(* Logix 5000 project; controller inz_PD_LK vendor 1 type 14 code 285 rev 34.11; software revision 34.01 *)

TASK MainTask (continuous, watchdog 500 ms) : Paleczka_silnik, Dzwonki_silnik, Paleczka_note_move, Dzwonki_belt_move, buttons, status, TIMER, Lights

MODULES
   Local : vendor 1 type 14 code 285 (5069 0, rev 34.11)
      serwowzmacniacz : vendor 1 type 45 code 1 (Ethernet 192.168.1.26, rev 5.2, AMotionDiagnostics RPI 1 ms)
      serwowzmacniacz2 : vendor 1 type 45 code 1 (Ethernet 192.168.1.27, rev 5.2, AMotionDiagnostics RPI 1 ms)
      Input : 5069-IB16 (5069 1, rev 2.1, StandardDataDriven RPI 5 ms)
      Output : 5069-OB16 (5069 2, rev 3.1, StandardDataDriven RPI 5 ms)
END_MODULES

VAR_GLOBAL   (* controller tags *)
   all_rise : BOOL;
   auto_mode : ALIAS FOR Local:1:I.Pt11.Data;
   belt_button : ALIAS FOR Local:1:I.Pt02.Data;
   belt_degree : DINT := 28;
   D_JOG_Axis_OFF : BOOL := 1;
   D_JOG_Axis_ON : BOOL;
   D_motor_start : BOOL;
   D_motor_stop : BOOL := 1;
   degree : DINT := -20;
   Dzwonki : AXIS_CIP_DRIVE;
   Estop_button : ALIAS FOR Local:1:I.Pt00.Data;
   forced_OFF : BOOL;
   forced_ON : BOOL := 1;
   green_lamp : ALIAS FOR Local:2:O.Pt13.Data;
   L_R_switch : ALIAS FOR Local:1:I.Pt10.Data;
   Motion : MOTION_GROUP;
   MotionControlMAFR_D : MOTION_INSTRUCTION := (FLAGS := 570425344, DN := 1, STATE := 1);
   MotionControlMAFR_P : MOTION_INSTRUCTION := (FLAGS := 570425344, DN := 1, STATE := 1);
   MotionControlMAJ_P : MOTION_INSTRUCTION := (FLAGS := 301989888, ER := 1, ERR := 5);
   MotionControlMAM : MOTION_INSTRUCTION := (FLAGS := 570425344, DN := 1);
   MotionControlMAM2 : MOTION_INSTRUCTION := (FLAGS := 704643072, DN := 1, PC := 1);
   MotionControlMAM3 : MOTION_INSTRUCTION := (FLAGS := 704643072, DN := 1, PC := 1);
   MotionControlMAM4 : MOTION_INSTRUCTION := (FLAGS := 704643072, DN := 1, PC := 1);
   MotionControlMAM5 : MOTION_INSTRUCTION := (FLAGS := 704643072, DN := 1, PC := 1);
   MotionControlMAS_D : MOTION_INSTRUCTION := (FLAGS := -1442840576, EN := 1, DN := 1, PC := 1);
   MotionControlMAS_P : MOTION_INSTRUCTION := (FLAGS := -1442840576, EN := 1, DN := 1, PC := 1);
   MotionControlOFF_D : MOTION_INSTRUCTION := (FLAGS := -1577058304, EN := 1, DN := 1, STATUS := 2, STATE := 1);
   MotionControlOFF_P : MOTION_INSTRUCTION := (FLAGS := -1577058304, EN := 1, DN := 1, STATUS := 2, STATE := 1);
   MotionControlON_D : MOTION_INSTRUCTION := (FLAGS := 570425344, DN := 1, STATE := 1);
   MotionControlON_P : MOTION_INSTRUCTION := (FLAGS := 570425344, DN := 1, STATE := 1);
   move_belt : BOOL;
   neg_belt_degree : DINT := -28;
   neg_degree : INT := 20;
   OSR_D_motor_start : BOOL;
   OSR_D_motor_stop : BOOL;
   OSR_forced_OFF : BOOL;
   OSR_forced_ON : BOOL;
   OSR_P_motor_start : BOOL;
   OSR_P_motor_stop : BOOL;
   OSR_start_now : BOOL;
   OSR_starting_ON : BOOL;
   P_JOG_Axis_OFF : BOOL := 1;
   P_JOG_Axis_ON : BOOL;
   P_motor_start : BOOL;
   P_motor_stop : BOOL := 1;
   Paleczka : AXIS_CIP_DRIVE;
   play_note : BOOL;
   play_note_rise : BOOL;
   PULSE_1Hz : BOOL;
   PULSE_2Hz : BOOL := 1;
   ready : BOOL;
   red_lamp : ALIAS FOR Local:2:O.Pt15.Data;
   reset : BOOL;
   reset_button : ALIAS FOR Local:1:I.Pt07.Data;
   stand_by : BOOL;
   start : BOOL; {access None}
   start_button : ALIAS FOR Local:1:I.Pt05.Data;
   start_degree : DINT := 20;
   start_now : BOOL;
   starting_ON : BOOL := 1;
   stop : BOOL := 1; {access None}
   switch_OFF : ALIAS FOR Local:1:I.Pt08.Data;
   switch_ON : ALIAS FOR Local:1:I.Pt09.Data;
   TIMER1N : TIMER := (PRE := 100);
   TIMER2N : TIMER := (PRE := 200);
   yellow_lamp : ALIAS FOR Local:2:O.Pt14.Data;
END_VAR

PROGRAM buttons   (* main routine buttons *)

ROUTINE buttons   (* ladder *)
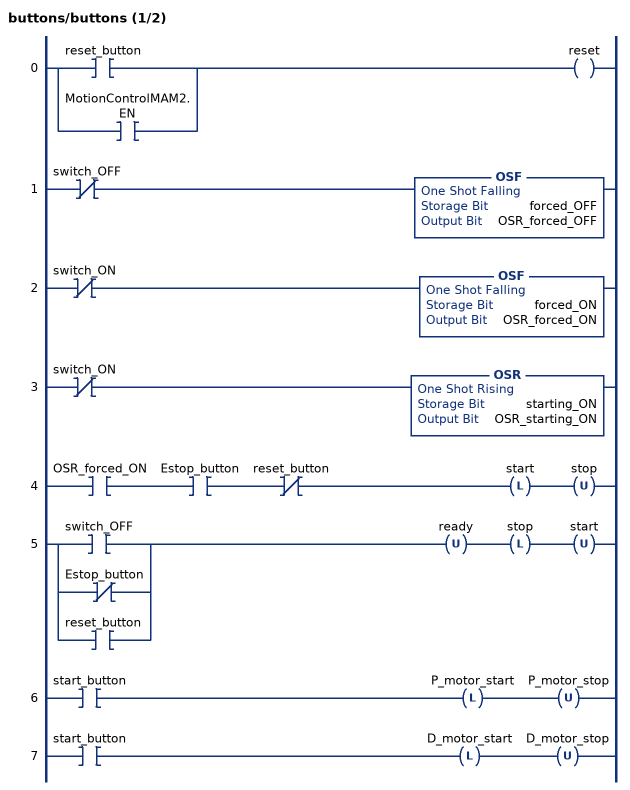
   0: [XIC(reset_button) ,XIC(MotionControlMAM2.EN) ]OTE(reset);
   1: XIO(switch_OFF)OSF(forced_OFF,OSR_forced_OFF);
   2: XIO(switch_ON)OSF(forced_ON,OSR_forced_ON);
   3: XIO(switch_ON)OSR(starting_ON,OSR_starting_ON);
   4: XIC(OSR_forced_ON)XIC(Estop_button)XIO(reset_button)OTL(start)OTU(stop);
   5: [XIC(switch_OFF) ,[XIO(Estop_button) ,XIC(reset_button) ] ]OTU(ready)OTL(stop)OTU(start);
   6: XIC(start_button)OTL(P_motor_start)OTU(P_motor_stop);
   7: XIC(start_button)OTL(D_motor_start)OTU(D_motor_stop);
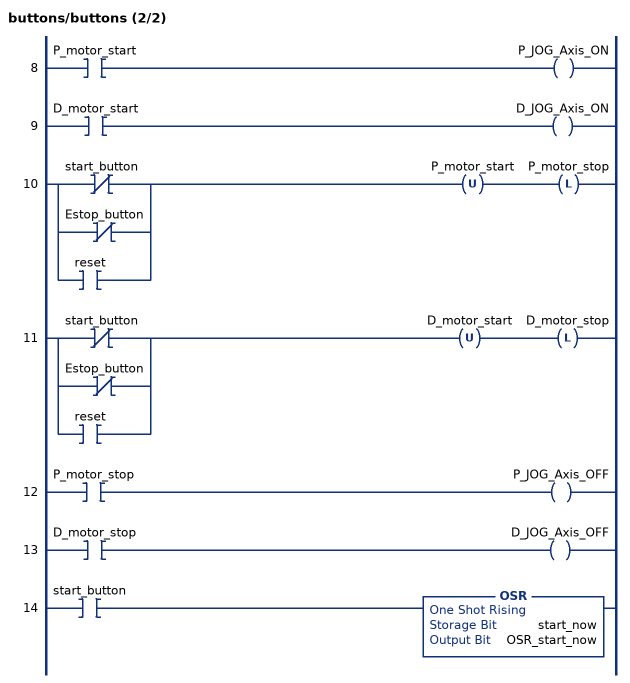
   8: XIC(P_motor_start)OTE(P_JOG_Axis_ON);
   9: XIC(D_motor_start)OTE(D_JOG_Axis_ON);
   10: [XIO(start_button) ,[XIO(Estop_button) ,XIC(reset) ] ]OTU(P_motor_start)OTL(P_motor_stop);
   11: [XIO(start_button) ,[XIO(Estop_button) ,XIC(reset) ] ]OTU(D_motor_start)OTL(D_motor_stop);
   12: XIC(P_motor_stop)OTE(P_JOG_Axis_OFF);
   13: XIC(D_motor_stop)OTE(D_JOG_Axis_OFF);
   14: XIC(start_button)OSR(start_now,OSR_start_now);
END_ROUTINE
END_PROGRAM

PROGRAM Dzwonki_belt_move   (* main routine belt_move *)

ROUTINE belt_move   (* ladder *)
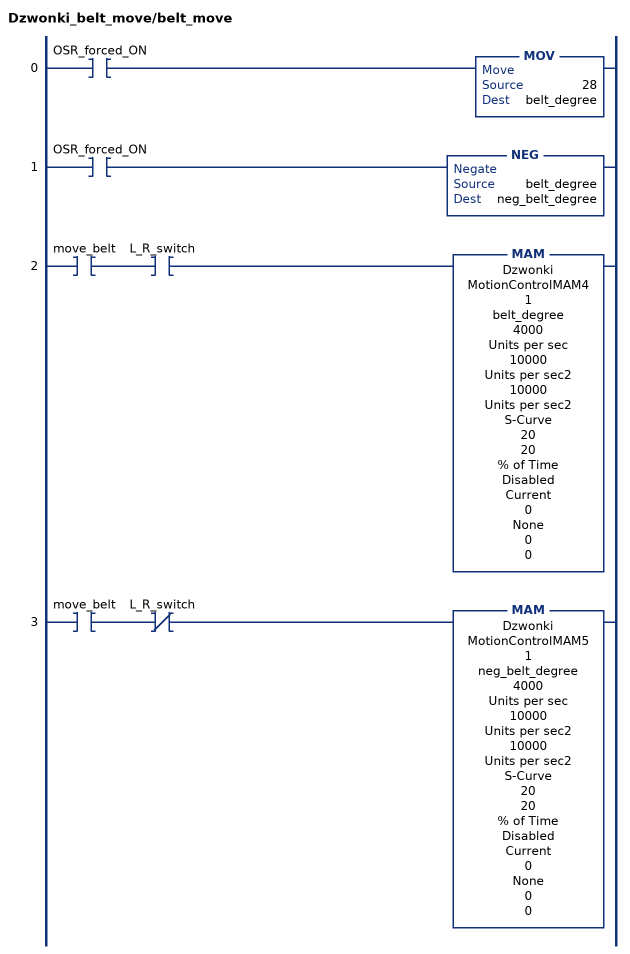
   0: XIC(OSR_forced_ON)MOV(28,belt_degree);
   1: XIC(OSR_forced_ON)NEG(belt_degree,neg_belt_degree);
   2: XIC(move_belt)XIC(L_R_switch)MAM(Dzwonki,MotionControlMAM4,1,belt_degree,4000,Units per sec,10000,Units per sec2,10000,Units per sec2,S-Curve,20,20,% of Time,Disabled,Current,0,None,0,0);
   3: XIC(move_belt)XIO(L_R_switch)MAM(Dzwonki,MotionControlMAM5,1,neg_belt_degree,4000,Units per sec,10000,Units per sec2,10000,Units per sec2,S-Curve,20,20,% of Time,Disabled,Current,0,None,0,0);
END_ROUTINE
END_PROGRAM

PROGRAM Dzwonki_silnik   (* main routine MainRoutine *)

ROUTINE MainRoutine   (* ladder *)
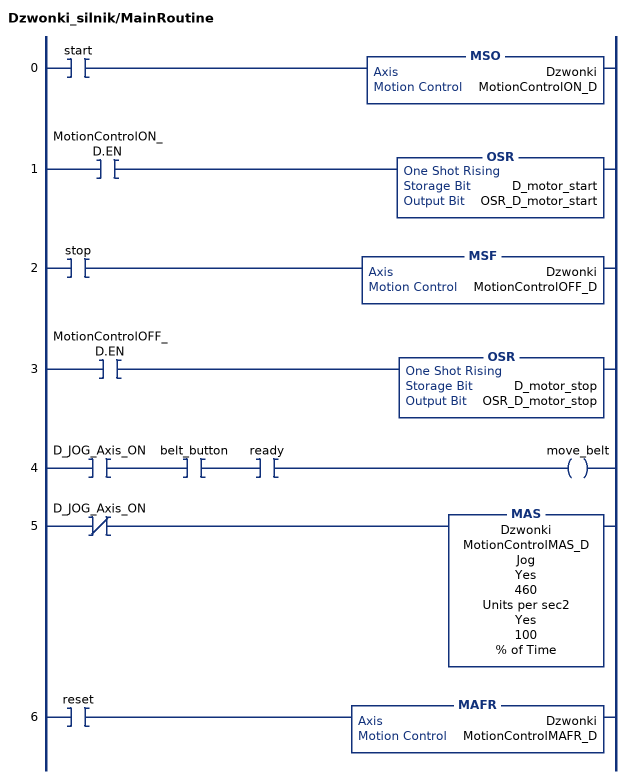
   0: XIC(start)MSO(Dzwonki,MotionControlON_D);
   1: XIC(MotionControlON_D.EN)OSR(D_motor_start,OSR_D_motor_start);
   2: XIC(stop)MSF(Dzwonki,MotionControlOFF_D);
   3: XIC(MotionControlOFF_D.EN)OSR(D_motor_stop,OSR_D_motor_stop);
   4: XIC(D_JOG_Axis_ON)XIC(belt_button)XIC(ready)OTE(move_belt);
   5: XIO(D_JOG_Axis_ON)MAS(Dzwonki,MotionControlMAS_D,Jog,Yes,460,Units per sec2,Yes,100,% of Time);
   6: XIC(reset)MAFR(Dzwonki,MotionControlMAFR_D);
END_ROUTINE
END_PROGRAM

PROGRAM Lights   (* main routine Lights *)

ROUTINE Lights   (* ladder *)
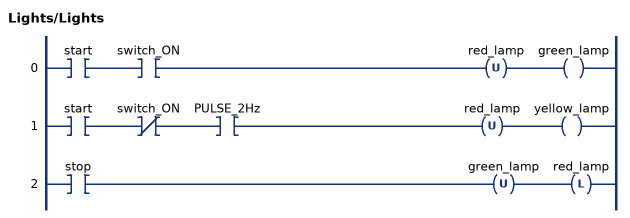
   0: XIC(start)XIC(switch_ON)OTU(red_lamp)OTE(green_lamp);
   1: XIC(start)XIO(switch_ON)XIC(PULSE_2Hz)OTU(red_lamp)OTE(yellow_lamp);
   2: XIC(stop)OTU(green_lamp)OTL(red_lamp);
END_ROUTINE
END_PROGRAM

PROGRAM Paleczka_note_move   (* main routine note_move *)

ROUTINE note_move   (* ladder *)
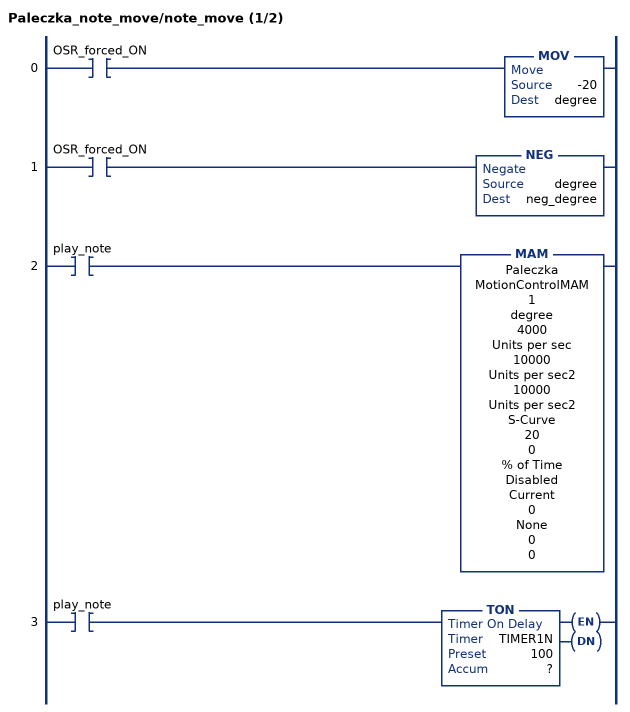
   0: XIC(OSR_forced_ON)MOV(-20,degree);
   1: XIC(OSR_forced_ON)NEG(degree,neg_degree);
   2: XIC(play_note)MAM(Paleczka,MotionControlMAM,1,degree,4000,Units per sec,10000,Units per sec2,10000,Units per sec2,S-Curve,20,0,% of Time,Disabled,Current,0,None,0,0);
   3: XIC(play_note)TON(TIMER1N,?,?);
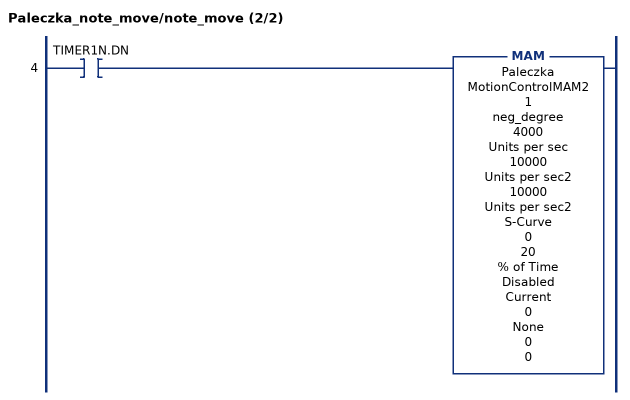
   4: XIC(TIMER1N.DN)MAM(Paleczka,MotionControlMAM2,1,neg_degree,4000,Units per sec,10000,Units per sec2,10000,Units per sec2,S-Curve,0,20,% of Time,Disabled,Current,0,None,0,0);
END_ROUTINE
END_PROGRAM

PROGRAM Paleczka_silnik   (* main routine MainRoutine *)

ROUTINE MainRoutine   (* ladder *)
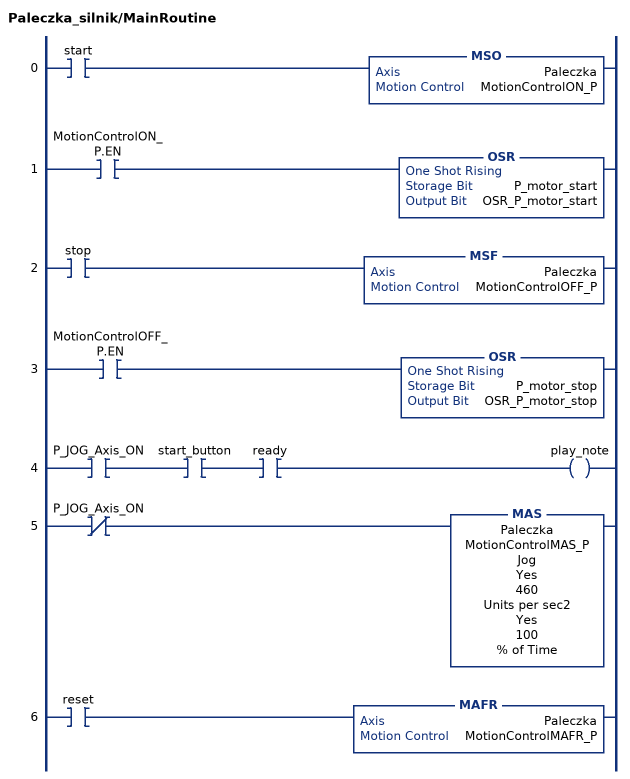
   0: XIC(start)MSO(Paleczka,MotionControlON_P);
   1: XIC(MotionControlON_P.EN)OSR(P_motor_start,OSR_P_motor_start);
   2: XIC(stop)MSF(Paleczka,MotionControlOFF_P);
   3: XIC(MotionControlOFF_P.EN)OSR(P_motor_stop,OSR_P_motor_stop);
   4: XIC(P_JOG_Axis_ON)XIC(start_button)XIC(ready)OTE(play_note);
   5: XIO(P_JOG_Axis_ON)MAS(Paleczka,MotionControlMAS_P,Jog,Yes,460,Units per sec2,Yes,100,% of Time);
   6: XIC(reset)MAFR(Paleczka,MotionControlMAFR_P);
END_ROUTINE
END_PROGRAM

PROGRAM status   (* main routine ready *)

ROUTINE ready   (* ladder *)
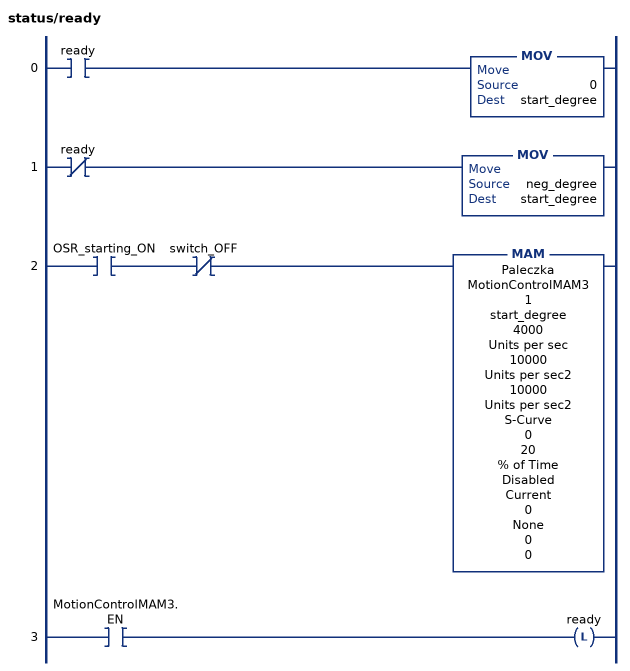
   0: XIC(ready)MOV(0,start_degree);
   1: XIO(ready)MOV(neg_degree,start_degree);
   2: XIC(OSR_starting_ON)XIO(switch_OFF)MAM(Paleczka,MotionControlMAM3,1,start_degree,4000,Units per sec,10000,Units per sec2,10000,Units per sec2,S-Curve,0,20,% of Time,Disabled,Current,0,None,0,0);
   3: XIC(MotionControlMAM3.EN)OTL(ready);
END_ROUTINE
END_PROGRAM

PROGRAM TIMER   (* main routine pulse *)
VAR
   TIMER1 : TIMER := (PRE := 1000, EN := 1, DN := 1);
   TIMER2 : TIMER := (PRE := 1000, ACC := 948, EN := 1, TT := 1);
   TIMER3 : TIMER := (PRE := 500, ACC := 448, TT := 1, DN := 1);
   TIMER4 : TIMER := (PRE := 500, ACC := 500, EN := 1, DN := 1);
END_VAR

ROUTINE pulse   (* ladder *)
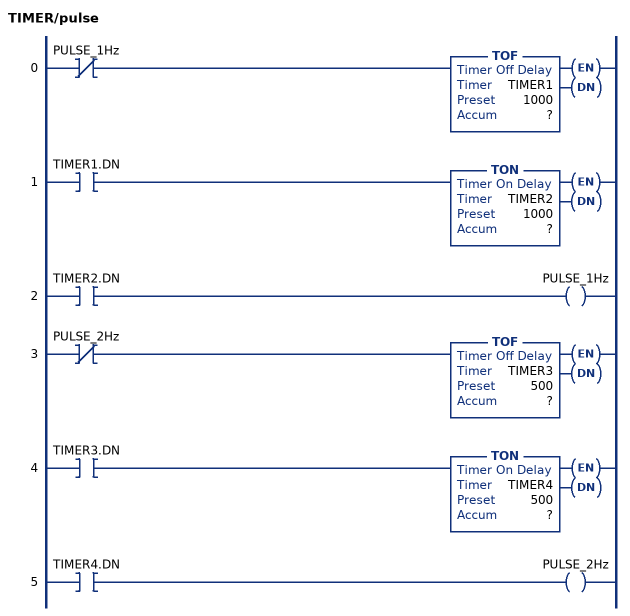
   0: XIO(PULSE_1Hz)TOF(TIMER1,?,?);
   1: XIC(TIMER1.DN)TON(TIMER2,?,?);
   2: XIC(TIMER2.DN)OTE(PULSE_1Hz);
   3: XIO(PULSE_2Hz)TOF(TIMER3,?,?);
   4: XIC(TIMER3.DN)TON(TIMER4,?,?);
   5: XIC(TIMER4.DN)OTE(PULSE_2Hz);
END_ROUTINE
END_PROGRAM
